FUNCTION F_DATE_RTN : DATE
VAR_INPUT
	stArg : ST_Arg;
END_VAR
VAR
	sysVar_Info : __SYSTEM.VAR_INFO;
END_VAR

sysVar_Info := __VARINFO(F_DATE_RTN);
IF stArg.TypeClass = sysVar_Info.TypeClass THEN 
	F_DATE_RTN := TO_DATE(stArg.sValue);
	END_IF

END_FUNCTION

(* stored: Version 1.1.0.1, ProductVersion 3.1.4024.4
   POU F_DATE_RTN: Id {e52b6963-e490-4e09-9635-36060138a765}, SpecialFunc None *)
